Fanuc TP program (LS listing): STRLOCAL.LS

/PROG  STRLOCAL
/ATTR
OWNER		= MNEDITOR;
COMMENT		= "StrLocal";
PROG_SIZE	= 0;
CREATE		= DATE 26-01-01  TIME 00:00:00;
MODIFIED	= DATE 26-01-01  TIME 00:00:00;
FILE_NAME	= ;
VERSION		= 0;
LINE_COUNT	= 7;
MEMORY_SIZE	= 0;
PROTECT		= READ_WRITE;
TCD:  STACK_SIZE	= 0,
      TASK_PRIORITY	= 50,
      TIME_SLICE	= 0,
      BUSY_LAMP_OFF	= 0,
      ABORT_REQUEST	= 0,
      PAUSE_REQUEST	= 0;
DEFAULT_GROUP	= 1,*,*,*,*;
CONTROL_CODE	= 00000000 00000000;
/MN
   1:  !RAPID StringProbe.StrLocal ;
   2:  CALL CA_TEXT(4,'X',0) ;
   3:  CALL CA_TEXT(4,'Y',1) ;
   4:  CALL CA_TEXT(25,'XY',0) ;
   5:  IF SR[4]<>SR[25],JMP LBL[1] ;
   6:  R[18:spLocal]=R[18:spLocal]+1    ;
   7:  LBL[1] ;
/POS
/END
